// TIA Portal V17 export
// export: Created 2025-03-07T09:19:34.5628616Z, ExportSetting WithDefaults, DisplayName Totally Integrated Automation Portal, DisplayVersion V17 Update 8, DisplayName TIA Portal Openness, DisplayVersion V17 Update 8, DisplayName TIA Portal Version Control Interface, DisplayVersion V17, DisplayName SINAMICS Startdrive Advanced, DisplayVersion V17 SP2, DisplayName SINAMICS Startdrive G110M, G120, G120C, G120D, G120P, G115D, DisplayVersion V17 SP2, DisplayName SINAMICS Startdrive G130, G150, S120, S150, SINAMICS MV, S210, DisplayVersion V17 SP2, DisplayName STEP 7 Professional, DisplayVersion V17 Update 8, DisplayName SINUMERIK ONE STEP 7 Toolbox, DisplayVersion V17 Update 12, DisplayName SINUMERIK 840D sl STEP 7 Toolbox, DisplayVersion V17 Update 12, DisplayName STEP 7 Safety, DisplayVersion V17 Update 6, DisplayName WinCC Advanced, DisplayVersion V17 Update 8
TYPE "LBP_typeModularMcpBaseOutput"
TITLE = Modular MCP image / Imagen de MCP modulares / Abbild modulare MCP
// Output image of base signals for modular MCP / Imagen de salida de señales base de MCP modulares / Ausgangsabbild von Basissignalen für modulare MCP
// stored: IsFailsafeCompliant false
   STRUCT
      optionalKey1 : Bool;   // Ausgangsabbild n+0 Bit 0; KT-OUT1 / output image n+0 bit 0; KT-OUT1 / Imagen de salida n+0 bit 0; KT-OUT1
      optionalKey2 : Bool;   // Ausgangsabbild n+0 Bit 1; KT-OUT2 / output image n+0 bit 1; KT-OUT2 / Imagen de salida n+0 bit 1; KT-OUT2
      optionalKey3 : Bool;   // Ausgangsabbild n+0 Bit 2; KT-OUT3 / output image n+0 bit 2; KT-OUT3 / Imagen de salida n+0 bit 2; KT-OUT3
      optionalKey4 : Bool;   // Ausgangsabbild n+0 Bit 3; KT-OUT4 / output image n+0 bit 3; KT-OUT4 / Imagen de salida n+0 bit 3; KT-OUT4
      optionalKey5 : Bool;   // Ausgangsabbild n+0 Bit 4; KT-OUT5 / output image n+0 bit 4; KT-OUT5 / Imagen de salida n+0 bit 4; KT-OUT5
      optionalKey6 : Bool;   // Ausgangsabbild n+0 Bit 5; KT-OUT6 / output image n+0 bit 5; KT-OUT6 / Imagen de salida n+0 bit 5; KT-OUT6
      optionalKey7 : Bool;   // Ausgangsabbild n+0 Bit 6; KT-OUT7 / output image n+0 bit 6; KT-OUT7 / Imagen de salida n+0 bit 6; KT-OUT7
      optionalKey8 : Bool;   // Ausgangsabbild n+0 Bit 7; KT-OUT8 / output image n+0 bit 7; KT-OUT8 / Imagen de salida n+0 bit 7; KT-OUT8
      optionalKey9 : Bool;   // Ausgangsabbild n+1 Bit 0; KT-OUT9 / output image n+1 bit 0; KT-OUT9 / Imagen de salida n+1 bit 0; KT-OUT9
      optionalKey10 : Bool;   // Ausgangsabbild n+1 Bit 1; KT-OUT10 / output image n+1 bit 1; KT-OUT10 / Imagen de salida n+1 bit 1; KT-OUT10
      optionalKey11 : Bool;   // Ausgangsabbild n+1 Bit 2; KT-OUT11 / output image n+1 bit 2; KT-OUT11 / Imagen de salida n+1 bit 2; KT-OUT11
      optionalKey12 : Bool;   // Ausgangsabbild n+1 Bit 3; KT-OUT12 / output image n+1 bit 3; KT-OUT12 / Imagen de salida n+1 bit 3; KT-OUT12
      optionalKey13 : Bool;   // Ausgangsabbild n+1 Bit 4; KT-OUT13 / output image n+1 bit 4; KT-OUT13 / Imagen de salida n+1 bit 4; KT-OUT13
      optionalKey14 : Bool;   // Ausgangsabbild n+1 Bit 5; KT-OUT14 / output image n+1 bit 5; KT-OUT14 / Imagen de salida n+1 bit 5; KT-OUT14
      optionalKey15 : Bool;   // Ausgangsabbild n+1 Bit 6; KT-OUT15 / output image n+1 bit 6; KT-OUT15 / Imagen de salida n+1 bit 6; KT-OUT15
      optionalKey16 : Bool;   // Ausgangsabbild n+1 Bit 7; KT-OUT16 / output image n+1 bit 7; KT-OUT16 / Imagen de salida n+1 bit 7; KT-OUT16
   END_STRUCT;
END_TYPE
